PROGRAM MAIN VAR _nCounter : UDINT; END_VAR

_nCounter := _nCounter + 1;
PRG_Syntax_Main();

END_PROGRAM

(* stored: Version 1.1.0.1, ProductVersion 3.1.4024.16
   POU MAIN: Id {d8471e9a-4c28-4033-bb92-e421a1f0a1c8}, SpecialFunc None *)
